// TIA Portal V18 export
ORGANIZATION_BLOCK "Main"   // OB1, FBD, ProgramCycle
TITLE = "Main Program Sweep (Cycle)"
{ S7_Optimized_Access := 'TRUE' }
// stored: SetENOAutomatically false
   VAR_INPUT
      Initial_Call : Bool;   // Initial call of this OB
      Remanence : Bool;   // =True, if remanent data are available
   END_VAR
   VAR_TEMP
      RET_VAL : Int;
      locTime : DTL;
   END_VAR
BEGIN

REGION Network 1: Inputs
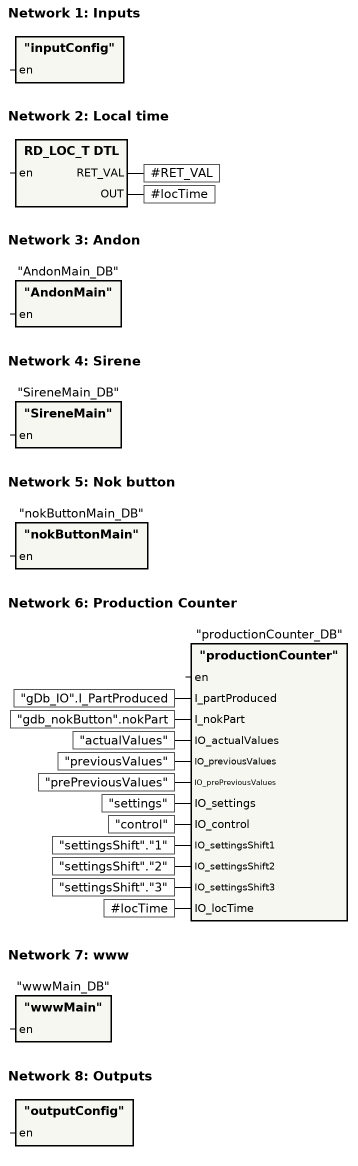
   "inputConfig"();
END_REGION

REGION Network 2: Local time
   #RET_VAL := RD_LOC_T(OUT => #locTime);
END_REGION

REGION Network 3: Andon
   "AndonMain_DB"();   // "AndonMain"
END_REGION

REGION Network 4: Sirene
   "SireneMain_DB"();   // "SireneMain"
END_REGION

REGION Network 5: Nok button
   "nokButtonMain_DB"();   // "nokButtonMain"
END_REGION

REGION Network 6: Production Counter
   "productionCounter_DB"(I_partProduced := "gDb_IO".I_PartProduced,   // "productionCounter"
                          I_nokPart := "gdb_nokButton".nokPart,
                          IO_actualValues := "actualValues",
                          IO_previousValues := "previousValues",
                          IO_prePreviousValues := "prePreviousValues",
                          IO_settings := "settings",
                          IO_control := "control",
                          IO_settingsShift1 := "settingsShift"."1",
                          IO_settingsShift2 := "settingsShift"."2",
                          IO_settingsShift3 := "settingsShift"."3",
                          IO_locTime := #locTime);
END_REGION

REGION Network 7: www
   "wwwMain_DB"();   // "wwwMain"
END_REGION

REGION Network 8: Outputs
   "outputConfig"();
END_REGION
END_ORGANIZATION_BLOCK
